# B&R Automation Studio project NewPendant_NG4_11_05_25A (part 5)

```c
	i = parCOOL_Tmo;
	strcpy(var[i].name , "Cool On/Off TimeOut");
	strcpy(var[i].enumTXT, "parCOOL_Tmo");
	var[i].PlcUnitIndx = unitIU;
	var[i].unitType = unitTime;
	var[i].DefaultUnit = UNIT_sec;
	var[i].precision = 1;
	cfg->Param[i].min = 0.0;
	cfg->Param[i].max = 5.0;
	cfg->Param[i].incrMin = 0.1;
	cfg->Param[i].incrMax = 1.0;
	cfg->Param[i].defaultVal = 3.0;
	var[i].segm = 0;

	///// INDX /////

	i = parINDX_StepDist;
	strcpy(var[i].name , "INDX Step Distance");
	strcpy(var[i].enumTXT, "parINDX_StepDist");
	var[i].PlcUnitIndx = unitIU;
	var[i].unitType = unitLength;
	var[i].DefaultUnit = UNIT_inch;
	var[i].precision = 1;
	cfg->Param[i].min = 0.0 * in_2_mm;
	cfg->Param[i].max = 200.0 * in_2_mm;
	cfg->Param[i].incrMin = 0.01 * in_2_mm;
	cfg->Param[i].incrMax = 1.0 * in_2_mm;
	cfg->Param[i].defaultVal = 4.5 * in_2_mm;
	var[i].segm = 0;

	i = parINDX_StepVel;
	strcpy(var[i].name , "INDX Step Vel");
	strcpy(var[i].enumTXT, "parINDX_StepVel");
	var[i].PlcUnitIndx = unitIU;
	var[i].unitType = unitPerc;
	var[i].DefaultUnit = UNIT_PERCENT;
	var[i].precision = 0;
	cfg->Param[i].min = 0.0;
	cfg->Param[i].max = 1.0;
	cfg->Param[i].incrMin = 0.01;
	cfg->Param[i].incrMax = 0.1;
	cfg->Param[i].defaultVal = 1.0;
	var[i].segm = 0;

	/*
	var[i].PlcUnitIndx = unitIU;
	var[i].unitType = unitSpeed;
	var[i].DefaultUnit = UNIT_inch_per_min;
	var[i].precision = 0;
	cfg->Param[i].min = 1.0 *  in_min_2_mm_s;
	cfg->Param[i].max = 10.0 *  in_min_2_mm_s;
	cfg->Param[i].incrMin = 0.1 * in_min_2_mm_s;
	cfg->Param[i].incrMax = 10.0 * cfg->Param[i].incrMin;
	cfg->Param[i].defaultVal = 3.0 * in_min_2_mm_s;
	var[i].segm = 0;
	*/

	i = parINDX_JogSpeedDirCntrl;
	strcpy(var[i].name , "INDX Jog Speed");
	strcpy(var[i].enumTXT, "parINDX_JogSpeedDirCntrl");
	var[i].PlcUnitIndx = unitIU;
	var[i].unitType = unitPerc;
	var[i].DefaultUnit = UNIT_PERCENT;
	var[i].precision = 0;
	cfg->Param[i].min = 0.0;
	cfg->Param[i].max = 1.0;
	cfg->Param[i].incrMin = 0.01;
	cfg->Param[i].incrMax = 0.1;
	cfg->Param[i].defaultVal = 1.0;
	var[i].segm = 0;

	i = parINDX_StepAfterBeats;
	strcpy(var[i].name , "Step After Beats");
	strcpy(var[i].enumTXT, "parINDX_StepAfterBeats");
	var[i].PlcUnitIndx = unitIU;
	var[i].unitType = unitIU;
	var[i].DefaultUnit = unitIU;
	var[i].precision = 0;
	cfg->Param[i].min = 0.0;
	cfg->Param[i].max = 99.0;
	cfg->Param[i].incrMin = 1.0;
	cfg->Param[i].incrMax = 1.0;
	cfg->Param[i].defaultVal = 0.0;
	var[i].segm = 0;

	//////  WRIST
	i = parWRST_JogSpeedDirCntrl;
	strcpy(var[i].name , "Weld Angle Jog Speed");
	strcpy(var[i].enumTXT, "parWRST_JogSpeedDirCntrl");
	var[i].PlcUnitIndx = unitIU;
	var[i].unitType = unitPerc;
	var[i].DefaultUnit = UNIT_PERCENT;
	var[i].precision = 1;
	cfg->Param[i].min = 0.0;
	cfg->Param[i].max = 1.0;
	cfg->Param[i].incrMin = 0.05;
	cfg->Param[i].incrMax = 0.1;
	cfg->Param[i].defaultVal = 0.75;
	var[i].segm = 0;

	//////  parTVL_POS_OFFSET
	i = parTVL_POS_OFFSET;
	strcpy(var[i].name , "TVL Pos Offset");
	strcpy(var[i].enumTXT, "parTVL_POS_OFFSET");
	var[i].PlcUnitIndx = unitIU;
	var[i].unitType = unitLength;
	var[i].DefaultUnit = UNIT_inch;
	var[i].precision = 1;
	cfg->Param[i].min = -200.0 * in_2_mm;
	cfg->Param[i].max = 200.0 * in_2_mm;
	cfg->Param[i].incrMin = 0.01 * in_2_mm;
	cfg->Param[i].incrMax = 1.0 * in_2_mm;
	cfg->Param[i].defaultVal = 0;
	var[i].segm = 0;

	i = parTVL_POS_PREDICT;
	strcpy(var[i].name , "TVL POS Predict Time");
	strcpy(var[i].enumTXT, "parTVL_POS_PREDICT");
	var[i].PlcUnitIndx = unitIU;
	var[i].unitType = unitTime;
	var[i].DefaultUnit = UNIT_sec;
	var[i].precision = 1;
	cfg->Param[i].min = 0.0;
	cfg->Param[i].max = 3.0;
	cfg->Param[i].incrMin = 0.1;
	cfg->Param[i].incrMax = 1.0;
	cfg->Param[i].defaultVal = 0.1;

	////////////////////////////////////

	i = parGEN_CalibDist;
	strcpy(var[i].name , "Calib Dist");
	strcpy(var[i].enumTXT, "parGEN_CalibDist");
	var[i].PlcUnitIndx = unitIU;
	var[i].unitType = unitLength;
	var[i].DefaultUnit = UNIT_inch;
	var[i].precision = 1;
	cfg->Param[i].min = 0.0;
	cfg->Param[i].max = 1000000;
	cfg->Param[i].incrMin = 0.254 *1;
	cfg->Param[i].incrMax = 25.4;
	cfg->Param[i].defaultVal = 0.0;
	var[i].segm = 0;

	i = parGEN_CalibDist_2;
	strcpy(var[i].name , "Calib Dist 2");
	strcpy(var[i].enumTXT, "parGEN_CalibDist_2");
	var[i].PlcUnitIndx = unitIU;
	var[i].unitType = unitLength;
	var[i].DefaultUnit = UNIT_inch;
	var[i].precision = 1;
	cfg->Param[i].min = 0.0;
	cfg->Param[i].max = 1000000;
	cfg->Param[i].incrMin = 0.254 *1;
	cfg->Param[i].incrMax = 25.4;
	cfg->Param[i].defaultVal = 0.0;
	var[i].segm = 0;

	i = parGEN_CalibDist1;
	strcpy(var[i].name , "Calib Dist1");
	strcpy(var[i].enumTXT, "parGEN_CalibDist1");
	var[i].PlcUnitIndx = unitIU;
	var[i].unitType = unitLength;
	var[i].DefaultUnit = UNIT_inch;
	var[i].precision = 1;
	cfg->Param[i].min = 0.0;
	cfg->Param[i].max = 1000000;
	cfg->Param[i].incrMin = 0.254 *1;
	cfg->Param[i].incrMax = 25.4;
	cfg->Param[i].defaultVal = 0.0;
	var[i].segm = 0;

	i = parGEN_CalibDist2;
	strcpy(var[i].name , "Calib Dist2");
	strcpy(var[i].enumTXT, "parGEN_CalibDist2");
	var[i].PlcUnitIndx = unitIU;
	var[i].unitType = unitLength;
	var[i].DefaultUnit = UNIT_inch;
	var[i].precision = 1;
	cfg->Param[i].min = 0.0;
	cfg->Param[i].max = 1000000;
	cfg->Param[i].incrMin = 0.254 *1;
	cfg->Param[i].incrMax = 25.4;
	cfg->Param[i].defaultVal = 0.0;
	var[i].segm = 0;

	i = parGEN_CalibDist3;
	strcpy(var[i].name , "Calib Dist3");
	strcpy(var[i].enumTXT, "parGEN_CalibDist3");
	var[i].PlcUnitIndx = unitIU;
	var[i].unitType = unitLength;
	var[i].DefaultUnit = UNIT_inch;
	var[i].precision = 1;
	cfg->Param[i].min = 0.0;
	cfg->Param[i].max = 1000000;
	cfg->Param[i].incrMin = 0.254 *1;
	cfg->Param[i].incrMax = 25.4;
	cfg->Param[i].defaultVal = 0.0;
	var[i].segm = 0;

	i = parGEN_CalibDist4;
	strcpy(var[i].name , "Calib Dist4");
	strcpy(var[i].enumTXT, "parGEN_CalibDist4");
	var[i].PlcUnitIndx = unitIU;
	var[i].unitType = unitLength;
	var[i].DefaultUnit = UNIT_inch;
	var[i].precision = 1;
	cfg->Param[i].min = 0.0;
	cfg->Param[i].max = 1000000;
	cfg->Param[i].incrMin = 0.254 *1;
	cfg->Param[i].incrMax = 25.4;
	cfg->Param[i].defaultVal = 0.0;
	var[i].segm = 0;

	i = parGEN_CalibTime;
	strcpy(var[i].name , "Calib Time");
	strcpy(var[i].enumTXT, "parGEN_CalibTime");
	var[i].PlcUnitIndx = unitIU;
	var[i].unitType = unitTime;
	var[i].DefaultUnit = UNIT_sec;
	var[i].precision = 1;
	cfg->Param[i].min = 0.0;
	cfg->Param[i].max = 1000000000.0;
	cfg->Param[i].incrMin = 0.05;
	cfg->Param[i].incrMax = 10.0;
	cfg->Param[i].defaultVal = 0.0;
	var[i].segm = 0;

	i = parGEN_CalibTime1;
	strcpy(var[i].name , "Calib Time1");
	strcpy(var[i].enumTXT, "parGEN_CalibTime1");
	var[i].PlcUnitIndx = unitIU;
	var[i].unitType = unitTime;
	var[i].DefaultUnit = UNIT_sec;
	var[i].precision = 1;
	cfg->Param[i].min = 0.0;
	cfg->Param[i].max = 1000000000.0;
	cfg->Param[i].incrMin = 0.05;
	cfg->Param[i].incrMax = 10.0;
	cfg->Param[i].defaultVal = 0.0;
	var[i].segm = 0;

	i = parGEN_CalibTime2;
	strcpy(var[i].name , "Calib Time2");
	strcpy(var[i].enumTXT, "parGEN_CalibTime2");
	var[i].PlcUnitIndx = unitIU;
	var[i].unitType = unitTime;
	var[i].DefaultUnit = UNIT_sec;
	var[i].precision = 1;
	cfg->Param[i].min = 0.0;
	cfg->Param[i].max = 1000000000.0;
	cfg->Param[i].incrMin = 0.05;
	cfg->Param[i].incrMax = 10.0;
	cfg->Param[i].defaultVal = 0.0;
	var[i].segm = 0;

	i = parGEN_CalibTime3;
	strcpy(var[i].name , "Calib Time3");
	strcpy(var[i].enumTXT, "parGEN_CalibTime3");
	var[i].PlcUnitIndx = unitIU;
	var[i].unitType = unitTime;
	var[i].DefaultUnit = UNIT_sec;
	var[i].precision = 1;
	cfg->Param[i].min = 0.0;
	cfg->Param[i].max = 1000000000.0;
	cfg->Param[i].incrMin = 0.05;
	cfg->Param[i].incrMax = 10.0;
	cfg->Param[i].defaultVal = 0.0;
	var[i].segm = 0;

	i = parGEN_CalibAmp1;
	strcpy(var[i].name , "GEN Calib Amp 1");
	strcpy(var[i].enumTXT, "parGEN_CalibAmp1");
	var[i].PlcUnitIndx = unitIU;
	var[i].unitType = unitAmp;
	var[i].DefaultUnit = UNIT_Amp;
	var[i].precision = 0;
	cfg->Param[i].min = 1.0;
	cfg->Param[i].max = 500.0;
	cfg->Param[i].incrMin = 1.0;
	cfg->Param[i].incrMax = 10.0;
	cfg->Param[i].defaultVal = 25.0;
	var[i].segm = 0;

	i = parGEN_CalibAmp2;
	strcpy(var[i].name , "GEN Calib Amp 2");
	strcpy(var[i].enumTXT, "parGEN_CalibAmp2");
	var[i].PlcUnitIndx = unitIU;
	var[i].unitType = unitAmp;
	var[i].DefaultUnit = UNIT_Amp;
	var[i].precision = 0;
	cfg->Param[i].min = 1.0;
	cfg->Param[i].max = 500.0;
	cfg->Param[i].incrMin = 1.0;
	cfg->Param[i].incrMax = 10.0;
	cfg->Param[i].defaultVal = 25.0;
	var[i].segm = 0;

	i = parGEN_CalibTime4;
	strcpy(var[i].name , "Calib Time4");
	strcpy(var[i].enumTXT, "parGEN_CalibTime4");
	var[i].PlcUnitIndx = unitIU;
	var[i].unitType = unitTime;
	var[i].DefaultUnit = UNIT_sec;
	var[i].precision = 1;
	cfg->Param[i].min = 0.0;
	cfg->Param[i].max = 1000000000.0;
	cfg->Param[i].incrMin = 0.05;
	cfg->Param[i].incrMax = 10.0;
	cfg->Param[i].defaultVal = 0.0;
	var[i].segm = 0;

	i = parGEN_AmpRead;
	strcpy(var[i].name , "Amp Meas.");
	strcpy(var[i].enumTXT, "parGEN_AmpRead");
	var[i].PlcUnitIndx = unitIU;
	var[i].unitType = unitAmp;
	var[i].DefaultUnit = UNIT_Amp;
	var[i].precision = 0;
	cfg->Param[i].min = 5.0;
	cfg->Param[i].max = 200.0;
	cfg->Param[i].incrMin = 1.0;
	cfg->Param[i].incrMax = 10.0;
	cfg->Param[i].defaultVal = 50.0;
	var[i].segm = 0;

	i = parGEN_WeldProgramRepeat;
	strcpy(var[i].name , "Weld Program Repeat");
	strcpy(var[i].enumTXT, "parGEN_WeldProgramRepeat");
	var[i].PlcUnitIndx = unitIU;
	var[i].unitType = unitIU;
	var[i].DefaultUnit = unitIU;
	var[i].precision = 0;
	cfg->Param[i].min = 0.0;
	cfg->Param[i].max = 99.0;
	cfg->Param[i].incrMin = 1.0;
	cfg->Param[i].incrMax = 1.0;
	cfg->Param[i].defaultVal = 0.0;
	var[i].segm = 0;

	i = parGEN_RadSpeed_Boost;
	strcpy(var[i].name , "TVL Radius Vel Boost");
	strcpy(var[i].enumTXT, "parGEN_RadSpeed_Boost");
	var[i].PlcUnitIndx = unitIU;
	var[i].unitType = unitPerc;
	var[i].DefaultUnit = UNIT_PERCENT;
	var[i].precision = 1;
	cfg->Param[i].min = 0.0;
	cfg->Param[i].max = 10.0;
	cfg->Param[i].incrMin = 0.05;
	cfg->Param[i].incrMax = 0.1;
	cfg->Param[i].defaultVal = 2.0;
	var[i].segm = 0;

	i = parGEN_Radius;
	strcpy(var[i].name , "Pole Radius");
	strcpy(var[i].enumTXT, "parGEN_Radius");
	var[i].PlcUnitIndx = unitIU;
	var[i].unitType = unitLength;
	var[i].DefaultUnit = UNIT_inch;
	var[i].precision = 1;
	cfg->Param[i].min = 0.0;
	cfg->Param[i].max = 1000000;
	cfg->Param[i].incrMin = 0.254 *1;
	cfg->Param[i].incrMax = 25.4;
	cfg->Param[i].defaultVal = 0.0;
	var[i].segm = 0;

	/////////////////////////////////////
	////////   Scaled variables

	i = varCurTVL_Vel;
	strcpy(var[i].enumTXT, "varCurTVL_Vel");
	strcpy(var[i].name , "TVL Vel 1FBK");
	var[i].pfVal = &Process[PROC_TVL].Fbk[0];
	strcpy(var[i].VarName , "Process[0].Fbk[0]");
	var[i].type = VAR_READONLY;
	var[i].PlcUnitIndx = unitIU;
	var[i].unitType = unitSpeed;
	var[i].DefaultUnit = UNIT_inch_per_min;
	var[i].precision = 0;

	i = varCurTVL_Vel_Calc;
	strcpy(var[i].enumTXT, "varCurTVL_Vel_Calc");
	strcpy(var[i].name , "TVL Vel FBK Calc");
	var[i].pfVal = &Process[PROC_TVL].Fbk[4];
	strcpy(var[i].VarName , "Process[0].Fbk[4]");
	var[i].type = VAR_READONLY;
	var[i].PlcUnitIndx = unitIU;
	var[i].unitType = unitSpeed;
	var[i].DefaultUnit = UNIT_inch_per_min;
	var[i].precision = 2;

	i = varTVL_Vel_Cmd;
	strcpy(var[i].enumTXT, "varTVL_Vel_Cmd");
	strcpy(var[i].name , "TVL Vel Cmd");
	var[i].pfVal = &Process[PROC_TVL].Fbk[1];
	strcpy(var[i].VarName , "Process[0].Fbk[1]");
	var[i].type = VAR_READONLY;
	var[i].PlcUnitIndx = unitIU;
	var[i].unitType = unitSpeed;
	var[i].DefaultUnit = UNIT_inch_per_min;
	var[i].precision = 0;

	i = varCurWF_Vel;
	strcpy(var[i].enumTXT, "varCurWF_Vel");
	strcpy(var[i].name , "WF Vel FBK");
	var[i].pfVal = &Process[PROC_WIRE_FEED].Fbk[0];
	strcpy(var[i].VarName , "Process[3].Fbk[0]");
	var[i].type = VAR_READONLY;
	var[i].PlcUnitIndx = unitIU;
	var[i].unitType = unitSpeed;
	var[i].DefaultUnit = UNIT_inch_per_min;
	var[i].precision = 0;

	i = varWF_Vel_Cmd;
	strcpy(var[i].enumTXT, "varWF_Vel_Cmd");
	strcpy(var[i].name , "WF Vel Cmd");
	var[i].pfVal = &Process[PROC_WIRE_FEED].Fbk[1];
	strcpy(var[i].VarName , "Process[3].Fbk[1]");
	var[i].type = VAR_READONLY;
	var[i].PlcUnitIndx = unitIU;
	var[i].unitType = unitSpeed;
	var[i].DefaultUnit = UNIT_inch_per_min;
	var[i].precision = 0;

	i = varCurWFDist;
	strcpy(var[i].enumTXT, "varCurWFDist");
	strcpy(var[i].name , "act WF Len");
	var[i].pfVal = &Process[PROC_WIRE_FEED].Fbk[4];
	strcpy(var[i].VarName , "Process[3].Fbk[4]");
	var[i].type = VAR_READONLY;
	var[i].PlcUnitIndx = unitIU;
	var[i].unitType = unitLength;
	var[i].DefaultUnit = UNIT_inch;
	var[i].precision = 0;

	i = varCurWP_Vel;
	strcpy(var[i].enumTXT, "varCurWP_Vel");
	strcpy(var[i].name , "WP Freq FBK");
	var[i].pfVal = &Process[PROC_WIRE_PULSE].Fbk[0];
	strcpy(var[i].VarName , "Process[4].Fbk[0]");
	var[i].type = VAR_READONLY;
	var[i].PlcUnitIndx = unitIU;
	var[i].unitType = unitFreq;
	var[i].DefaultUnit = UNIT_Hz;
	var[i].precision = 1;

	i = varWP_Vel_Cmd;
	strcpy(var[i].enumTXT, "varWP_Vel_Cmd");
	strcpy(var[i].name , "WP Freq Cmd");
	var[i].pfVal = &Process[PROC_WIRE_PULSE].Fbk[1];
	strcpy(var[i].VarName , "Process[4].Fbk[1]");
	var[i].type = VAR_READONLY;
	var[i].PlcUnitIndx = unitIU;
	var[i].unitType = unitFreq;
	var[i].DefaultUnit = UNIT_Hz;
	var[i].precision = 1;

	i = varCurArc_Volt;
	strcpy(var[i].enumTXT, "varCurArc_Volt");
	strcpy(var[i].name , "Arc Volt FBK");
	var[i].pfVal = &Process[PROC_AVC].Fbk[0];
	strcpy(var[i].VarName , "Process[2].Fbk[0]");
	var[i].type = VAR_READONLY;
	var[i].PlcUnitIndx = unitIU;
	var[i].unitType = unitVolt;
	var[i].DefaultUnit = UNIT_Volt;
	var[i].precision = 1;

	i = varArc_Volt_Cmd;
	strcpy(var[i].enumTXT, "varArc_Volt_Cmd");
	strcpy(var[i].name , "Arc Volt Cmd");
	var[i].pfVal = &Process[PROC_AVC].Fbk[1];
	strcpy(var[i].VarName , "Process[2].Fbk[1]");
	var[i].type = VAR_READONLY;
	var[i].PlcUnitIndx = unitIU;
	var[i].unitType = unitVolt;
	var[i].DefaultUnit = UNIT_Volt;
	var[i].precision = 1;

	i = varCurTIG_Amp;
	strcpy(var[i].enumTXT, "varCurTIG_Amp");
	strcpy(var[i].name , "TIG Amp FBK");
	var[i].pfVal = &Process[PROC_TIG_PS].Fbk[0];
	strcpy(var[i].VarName , "Process[5].Fbk[0]");
	var[i].type = VAR_READONLY;
	var[i].PlcUnitIndx = unitIU;
	var[i].unitType = unitAmp;
	var[i].DefaultUnit = UNIT_Amp;
	var[i].precision = 1;

	i = varTIG_Amp_Cmd;
	strcpy(var[i].enumTXT, "varTIG_Amp_Cmd");
	strcpy(var[i].name , "TIG Amp CMD");
	var[i].pfVal = &Process[PROC_TIG_PS].Fbk[1];
	strcpy(var[i].VarName , "Process[5].Fbk[1]");
	var[i].type = VAR_READONLY;
	var[i].PlcUnitIndx = unitIU;
	var[i].unitType = unitAmp;
	var[i].DefaultUnit = UNIT_Amp;
	var[i].precision = 0;

	i = varCurHW_Amp;
	strcpy(var[i].enumTXT, "varCurHW_Amp");
	strcpy(var[i].name , "HW Amp FBK");
	var[i].pfVal = &Process[PROC_HW_PS].Fbk[0];
	strcpy(var[i].VarName , "Process[6].Fbk[0]");
	var[i].type = VAR_READONLY;
	var[i].PlcUnitIndx = unitIU;
	var[i].unitType = unitAmp;
	var[i].DefaultUnit = UNIT_Amp;
	var[i].precision = 0;

	i = varHW_Amp_Cmd;
	strcpy(var[i].enumTXT, "varHW_Amp_Cmd");
	strcpy(var[i].name , "HW Amp CMD");
	var[i].pfVal = &Process[PROC_HW_PS].Fbk[1];
	strcpy(var[i].VarName , "Process[6].Fbk[1]");
	var[i].type = VAR_READONLY;
	var[i].PlcUnitIndx = unitIU;
	var[i].unitType = unitAmp;
	var[i].DefaultUnit = UNIT_Amp;
	var[i].precision = 0;

	i = varCurHW_Volt; // new
	strcpy(var[i].enumTXT, "varCurHW_Volt");
	strcpy(var[i].name , "HW Volt FBK");
	var[i].pfVal = &Process[PROC_HW_PS].Fbk[2];
	strcpy(var[i].VarName , "Process[6].Fbk[2]");
	var[i].type = VAR_READONLY;
	var[i].PlcUnitIndx = unitIU;
	var[i].unitType = unitVolt;
	var[i].DefaultUnit = UNIT_Volt;
	var[i].precision = 1;

	i = varHW_Volt_Cmd; // new
	strcpy(var[i].enumTXT, "varHW_Volt_Cmd");
	strcpy(var[i].name , "HW Volt CMD");
	var[i].pfVal = &Process[PROC_HW_PS].Fbk[3];
	strcpy(var[i].VarName , "Process[6].Fbk[3]");
	var[i].type = VAR_READONLY;
	var[i].PlcUnitIndx = unitIU;
	var[i].unitType = unitVolt;
	var[i].DefaultUnit = UNIT_Volt;
	var[i].precision = 1;

	i = varOSC_CurPos;
	strcpy(var[i].enumTXT, "varOSC_CurPos");
	strcpy(var[i].name , "act OSC Pos");
	var[i].pfVal = &Process[PROC_OSC].Fbk[0];
	strcpy(var[i].VarName , "Process[1].Fbk[0]");
	var[i].type = VAR_READONLY;
	var[i].PlcUnitIndx = unitIU;
	var[i].unitType = unitLength;
	var[i].DefaultUnit = UNIT_inch;
	var[i].precision = 1;

	i = varOSC_Centr;
	strcpy(var[i].enumTXT, "varOSC_Centr");
	strcpy(var[i].name , "act OSC Centr");
	var[i].pfVal = &Process[PROC_OSC].Fbk[1];
	strcpy(var[i].VarName , "Process[1].Fbk[1]");
	var[i].type = VAR_READONLY;
	var[i].PlcUnitIndx = unitIU;
	var[i].unitType = unitLength;
	var[i].DefaultUnit = UNIT_inch;
	var[i].precision = 1;

	i = varOSC_CurRawPos;
	strcpy(var[i].enumTXT, "varOSC_CurRawPos");
	strcpy(var[i].name , "act OSC Pos");
	var[i].pfVal = &Process[PROC_OSC].Fbk[2];
	strcpy(var[i].VarName , "Process[1].Fbk[2]");
	var[i].type = VAR_READONLY;
	var[i].PlcUnitIndx = unitIU;
	var[i].unitType = unitLength;
	var[i].DefaultUnit = UNIT_inch;
	var[i].precision = 2;

	i = varOSC_Amplit_Cmd;
	strcpy(var[i].enumTXT, "varOSC_Amplit_Cmd");
	strcpy(var[i].name , "OSC Amplit Cmd");
	var[i].pfVal = &Process[PROC_OSC].Fbk[3];
	strcpy(var[i].VarName , "Process[1].Fbk[3]");
	var[i].type = VAR_READONLY;
	var[i].PlcUnitIndx = unitIU;
	var[i].unitType = unitLength;
	var[i].DefaultUnit = UNIT_inch;
	var[i].precision = 1;

	i = varOSC_curExcurTm;
	strcpy(var[i].enumTXT, "varOSC_curExcurTm");
	strcpy(var[i].name , "act Excur Tm");
	var[i].pfVal = &Process[PROC_OSC].Fbk[4];
	strcpy(var[i].VarName , "Process[1].Fbk[4]");
	var[i].type = VAR_READONLY;
	var[i].PlcUnitIndx = unitIU;
	var[i].unitType = unitTime;
	var[i].DefaultUnit = UNIT_sec;
	var[i].precision = 1;

	i = varOSC_ExcurTm_Cmd;
	strcpy(var[i].enumTXT, "varOSC_ExcurTm_Cmd");
	strcpy(var[i].name , "OSC Excur Tm Cmd");
	var[i].pfVal = &Process[PROC_OSC].Fbk[5];
	strcpy(var[i].VarName , "Process[1].Fbk[5]");
	var[i].type = VAR_READONLY;
	var[i].PlcUnitIndx = unitIU;
	var[i].unitType = unitTime;
	var[i].DefaultUnit = UNIT_sec;
	var[i].precision = 1;

	i = varOSC_Dwell_In_Cmd;
	strcpy(var[i].enumTXT, "varOSC_Dwell_In_Cmd");
	strcpy(var[i].name , "varOSC Dwell In Cmd");
	var[i].pfVal = &Process[PROC_OSC].Fbk[6];
	strcpy(var[i].VarName , "Process[1].Fbk[6]");
	var[i].type = VAR_READONLY;
	var[i].PlcUnitIndx = unitIU;
	var[i].unitType = unitTime;
	var[i].DefaultUnit = UNIT_sec;
	var[i].precision = 1;

	i = varOSC_Dwell_Out_Cmd;
	strcpy(var[i].enumTXT, "varOSC_Dwell_Out_Cmd");
	strcpy(var[i].name , "Dwell_Out_Cmd Cmd");
	var[i].pfVal = &Process[PROC_OSC].Fbk[7];
	strcpy(var[i].VarName , "Process[1].Fbk[7]");
	var[i].type = VAR_READONLY;
	var[i].PlcUnitIndx = unitIU;
	var[i].unitType = unitTime;
	var[i].DefaultUnit = UNIT_sec;
	var[i].precision = 1;

	i = varINDX_A_Pos;
	strcpy(var[i].enumTXT, "varINDX_A_Pos");
	strcpy(var[i].name , "act Indx A Pos");
	var[i].pfVal = &Process[PROC_INDX].Fbk[0];
	strcpy(var[i].VarName , "Process[10].Fbk[0]");
	var[i].type = VAR_READONLY;
	var[i].PlcUnitIndx = unitIU;
	var[i].unitType = unitLength;
	var[i].DefaultUnit = UNIT_inch;
	var[i].precision = 2;

	i = varINDX_B_Pos;
	strcpy(var[i].enumTXT, "varINDX_B_Pos");
	strcpy(var[i].name , "act Indx B Pos");
	var[i].pfVal = &Process[PROC_INDX].Fbk[1];
	strcpy(var[i].VarName , "Process[10].Fbk[1]");
	var[i].type = VAR_READONLY;
	var[i].PlcUnitIndx = unitIU;
	var[i].unitType = unitLength;
	var[i].DefaultUnit = UNIT_inch;
	var[i].precision = 2;

	i = varINDX_Dif_Pos;
	strcpy(var[i].enumTXT, "varINDX_Dif_Pos");
	strcpy(var[i].name , "act Indx Dif Pos");
	var[i].pfVal = &Process[PROC_INDX].Fbk[2];
	strcpy(var[i].VarName , "Process[10].Fbk[2]");
	var[i].type = VAR_READONLY;
	var[i].PlcUnitIndx = unitIU;
	var[i].unitType = unitLength;
	var[i].DefaultUnit = UNIT_inch;
	var[i].precision = 3;

	i = varGlobTimer;
	strcpy(var[i].enumTXT, "varGlobTimer");
	strcpy(var[i].name , "Timer");
	var[i].pfVal = &GlobalTimer;
	strcpy(var[i].VarName , "GlobalTimer");
	var[i].type = VAR_READONLY;
	var[i].PlcUnitIndx = unitIU;
	var[i].unitType = unitTime;
	var[i].DefaultUnit = UNIT_sec;
	var[i].precision = 0;

	////////////////////////////

	i = parENUM_OSC_CAM;
	strcpy(cfg->EnumVar[i].enumTXT , "parENUM_OSC_CAM");
	strcpy(cfg->EnumVar[i].name , "OSC Cam Type ");
	cfg->EnumVar[i].TxtIndx = resTXT_OSC_CAM;
	cfg->EnumVar[i].segm = 0;
	cfg->Param_ENUM[i].defaultVal = 1;
	cfg->Param_ENUM[i].min = 0;
	cfg->Param_ENUM[i].max = CAM_NUM-1;

	i = parENUM_WeldProgramLinkMode;
	strcpy(cfg->EnumVar[i].enumTXT , "parENUM_WeldProgramLinkMode");
	strcpy(cfg->EnumVar[i].name , "Load Next Program ");
	cfg->EnumVar[i].TxtIndx = resWelProgramLinkMode;
	cfg->EnumVar[i].segm = 0;
	cfg->Param_ENUM[i].defaultVal = 0;
	cfg->Param_ENUM[i].min = 0;
	cfg->Param_ENUM[i].max = 1;

	i= parENUM_PathMode;
	strcpy(cfg->EnumVar[i].enumTXT , "parENUM_PathMode");
	strcpy(cfg->EnumVar[i].name , "Change Head at the end ");
	cfg->EnumVar[i].TxtIndx = resPathMode;
	cfg->EnumVar[i].segm = 0;
	cfg->Param_ENUM[i].defaultVal = 0;
	cfg->Param_ENUM[i].min = 0;
	cfg->Param_ENUM[i].max = 1;

	i= parENUM_TVL_MODE;
	strcpy(cfg->EnumVar[i].enumTXT , "parENUM_TVL_MODE");
	strcpy(cfg->EnumVar[i].name , "TVL Enc Mode");
	cfg->EnumVar[i].TxtIndx = resTVLMode;
	cfg->EnumVar[i].segm = 0;
	cfg->Param_ENUM[i].defaultVal = 0;
	cfg->Param_ENUM[i].min = 0;
	cfg->Param_ENUM[i].max = 3;

	i= parENUM_TVL_SYN_MODE;
	strcpy(cfg->EnumVar[i].enumTXT , "parENUM_TVL_SYN_MODE");
	strcpy(cfg->EnumVar[i].name , "TVL Synch Mode");
	cfg->EnumVar[i].TxtIndx = resSYNCOption; // Chris add this parameter to enum
	cfg->EnumVar[i].segm = 0;
	cfg->Param_ENUM[i].defaultVal = 0;
	cfg->Param_ENUM[i].min = 0;
	cfg->Param_ENUM[i].max = 2;

	i= parENUM_WF_SYN_MODE;
	strcpy(cfg->EnumVar[i].enumTXT , "parENUM_WF_SYN_MODE");
	strcpy(cfg->EnumVar[i].name , "WF Synch Mode");
	cfg->EnumVar[i].TxtIndx = resSYNCOption;
	cfg->EnumVar[i].segm = 0;
	cfg->Param_ENUM[i].defaultVal = 0;
	cfg->Param_ENUM[i].min = 0;
	cfg->Param_ENUM[i].max = 2;

	i= parENUM_WP_SYN_MODE;
	strcpy(cfg->EnumVar[i].enumTXT , "parENUM_WP_SYN_MODE");
	strcpy(cfg->EnumVar[i].name , "WP Synch Mode");
	cfg->EnumVar[i].TxtIndx = resSYNCOption;
	cfg->EnumVar[i].segm = 0;
	cfg->Param_ENUM[i].defaultVal = 0;
	cfg->Param_ENUM[i].min = 0;
	cfg->Param_ENUM[i].max = 2;

	/*
	i = parENUM_WeldProgramCase;
	strcpy(cfg->EnumVar[i].enumTXT , ""); // Use as a spare
	//strcpy(cfg->EnumVar[i].enumTXT , "parENUM_WeldProgramCase");
	cfg->EnumVar[i].TxtIndx = resWeldProgramCase;
	cfg->EnumVar[i].segm = 0;
	cfg->Param_ENUM[i].defaultVal = 0;
	cfg->Param_ENUM[i].min = 0;
	cfg->Param_ENUM[i].max = 5;
	*/

	i = parENUM_AVC_Mode;
	strcpy(cfg->EnumVar[i].enumTXT , "parENUM_AVC_Mode");
	strcpy(cfg->EnumVar[i].name , "AVC Type ");
	cfg->EnumVar[i].TxtIndx = resAVCMode;
	cfg->EnumVar[i].segm = 0;
	cfg->Param_ENUM[i].defaultVal = 0;
	cfg->Param_ENUM[i].min = 0;
	cfg->Param_ENUM[i].max = 3;

	i = parENUM_TIG_Mode;
	strcpy(cfg->EnumVar[i].enumTXT , "parENUM_TIG_Mode");
	strcpy(cfg->EnumVar[i].name , "TIG PS Mode ");
	cfg->EnumVar[i].TxtIndx = resTIGMode;
	cfg->EnumVar[i].segm = 0;
	cfg->Param_ENUM[i].defaultVal = 0;
	cfg->Param_ENUM[i].min = 0;
	cfg->Param_ENUM[i].max = 3;

	i = parENUM_TIG_Cal_Mode;
	strcpy(cfg->EnumVar[i].enumTXT , "parENUM_TIG_Cal_Mode");
	strcpy(cfg->EnumVar[i].name , "TIG PS Cal. Mode ");
	cfg->EnumVar[i].TxtIndx = resTigCalMode;
	cfg->EnumVar[i].segm = 0;
	cfg->Param_ENUM[i].defaultVal = 0;
	cfg->Param_ENUM[i].min = 0;
	cfg->Param_ENUM[i].max = 1;

	i = parENUM_WF_WP_Relation;
	strcpy(cfg->EnumVar[i].enumTXT , "parENUM_WF_WP_Relation");
	strcpy(cfg->EnumVar[i].name , "Relation between WF and WP");
	cfg->EnumVar[i].TxtIndx = resTXT_ON_OFF;
	cfg->EnumVar[i].segm = 0;
	cfg->Param_ENUM[i].defaultVal = 0;
	cfg->Param_ENUM[i].min = 0;
	cfg->Param_ENUM[i].max = 1;

	i = parENUM_ARCLINK_MODE;
	strcpy(cfg->EnumVar[i].enumTXT , "parENUM_ARCLINK_MODE");
	strcpy(cfg->EnumVar[i].name , "ARcLink ");
	cfg->EnumVar[i].TxtIndx = resTXT_ON_OFF;
	cfg->EnumVar[i].segm = 0;
	cfg->Param_ENUM[i].defaultVal = 0;
	cfg->Param_ENUM[i].min = 0;
	cfg->Param_ENUM[i].max = 1;

	i = parENUM_OSC_Mode;
	strcpy(cfg->EnumVar[i].enumTXT , "parENUM_OSC_Mode");
	strcpy(cfg->EnumVar[i].name , "OSC Mode ");
	cfg->EnumVar[i].TxtIndx = resTXT_OSC_Mode;
	cfg->EnumVar[i].segm = 0;
	cfg->Param_ENUM[i].defaultVal = 0;
	cfg->Param_ENUM[i].min = 0;
	cfg->Param_ENUM[i].max = 3;

	i = parENUM_OSC_Synch;
	strcpy(cfg->EnumVar[i].enumTXT , "parENUM_OSC_Synch");
	strcpy(cfg->EnumVar[i].name , "OSC Indx Synch ");
	cfg->EnumVar[i].TxtIndx = resTXT_OSC_Synch;
	cfg->EnumVar[i].segm = 0;
	cfg->Param_ENUM[i].defaultVal = 0;
	cfg->Param_ENUM[i].min = 0;
	cfg->Param_ENUM[i].max = 4;

	i = parENUM_WF_AUX;
	strcpy(cfg->EnumVar[i].enumTXT , "parENUM_WF_AUX");
	strcpy(cfg->EnumVar[i].name , "parENUM_WF_AUX");
	cfg->EnumVar[i].TxtIndx = resTXT_WF_AUX;
	cfg->EnumVar[i].segm = 0;
	cfg->Param_ENUM[i].defaultVal = 0;
	cfg->Param_ENUM[i].min = 0;
	cfg->Param_ENUM[i].max = 2;

	///////Int Variable    //////////

	i = parINT_NumZone;
	strcpy(cfg->IntVar[i].enumTXT , "parINT_NumZone");
	strcpy(cfg->IntVar[i].name , 	"Segments per Travel");
	cfg->IntVar[i].pVal = &curCfg->Param_INT[parINT_NumZone].val[0];
	strcpy(cfg->IntVar[i].VarName , "CurCfg.Param_INT[0].val[0]"); //this is for Android
	cfg->IntVar[i].DefaultVal = 1;
	cfg->IntVar[i].Min = 1;
	cfg->IntVar[i].Max = 1000;
	cfg->IntVar[i].segm = 0;

	i = varINT_PIN_PER_ROT;
	strcpy(cfg->IntVar[i].enumTXT , "varINT_PIN_PER_ROT");
	strcpy(cfg->IntVar[i].name , 	"Pins per 360 degree");
	cfg->IntVar[i].pVal = &calib->GenSetup[SETUP_PIN_PER_ROT];
	strcpy(cfg->IntVar[i].VarName , "CurCalib.GenSetup[0]"); //this is for Android
	cfg->IntVar[i].Min = 1;
	cfg->IntVar[i].Max = 1000;

	i = varINT_SEGM_NO;
	strcpy(cfg->IntVar[i].enumTXT , "varINT_SEGM_NO");
	strcpy(cfg->IntVar[i].name , 	"Segments Number");
	cfg->IntVar[i].pVal = &calib->GenSetup[SETUP_SEGM_NO];
	strcpy(cfg->IntVar[i].VarName , "CurCalib.GenSetup[1]"); //this is for Android
	cfg->IntVar[i].Min = 1;
	cfg->IntVar[i].Max = 1000;

	/*
	i = varINT_ZONE_NO;
	strcpy(cfg->IntVar[i].enumTXT , "varINT_ZONE_NO");
	cfg->IntVar[i].pVal = &calib->GenSetup[SETUP_ZONE_NO];
	strcpy(cfg->IntVar[i].VarName , "CurCalib.GenSetup[2]"); //this is for Android
	cfg->IntVar[i].Min = 1;
	cfg->IntVar[i].Max = 1000;

	i= varINT_curSegm;
	strcpy(cfg->IntVar[i].enumTXT , "varINT_curSegm");
	strcpy(cfg->IntVar[i].name , 	"Current Pin");
	cfg->IntVar[i].pVal = &m->curSegm[HEAD_SEGM];
	strcpy(cfg->IntVar[i].VarName , "Master[0].curSegm[3]"); //this is for Android
	cfg->IntVar[i].Min = 1;
	cfg->IntVar[i].Max = 1000;
	*/

	i = varINT_curZone;
	strcpy(cfg->IntVar[i].enumTXT , "varINT_curZone");
	strcpy(cfg->IntVar[i].name , 	"Current Segment");
	cfg->IntVar[i].pVal = &m->curSegm[ZONE];
	strcpy(cfg->IntVar[i].VarName , "Master[0].curSegm[1]"); //this is for Android
	cfg->IntVar[i].Min = 1;
	cfg->IntVar[i].Max = 1000;

	i = varINT_StartPos;
	strcpy(cfg->IntVar[i].enumTXT , "varINT_StartPos");
	strcpy(cfg->IntVar[i].name , 	"Start Position");
	cfg->IntVar[i].pVal = &StartPos;
	strcpy(cfg->IntVar[i].VarName , "StartPos"); //this is for Android
	cfg->IntVar[i].Min = -32767;
	cfg->IntVar[i].Max = 32767;

	i = varINT_FinalPos;
	strcpy(cfg->IntVar[i].enumTXT , "varINT_FinalPos");
	strcpy(cfg->IntVar[i].name , 	"Target Position");
	cfg->IntVar[i].pVal = &FinalPos;
	strcpy(cfg->IntVar[i].VarName , "FinalPos"); //this is for Android
	cfg->IntVar[i].Min = -32767;
	cfg->IntVar[i].Max = 32767;

	i = varINT_CurTVLPos;
	strcpy(cfg->IntVar[i].enumTXT , "varINT_CurTVLPos");
	strcpy(cfg->IntVar[i].name , 	"Current TVL Position");
	cfg->IntVar[i].pVal = &m->curSegm[ACT_TVL_DIST];
	strcpy(cfg->IntVar[i].VarName , "Master[0].curSegm[4]"); //this is for Android
	cfg->IntVar[i].Min = -32767;
	cfg->IntVar[i].Max = 32767;

	/// Strings
	i = parSTRING_FreeTXT;
	strcpy(cfg->StringVar[i].enumTXT , "parSTRING_FreeTXT");
	strcpy(cfg->StringVar[i].name, "FreeText");
	cfg->Param_STR[i].len = 5;
	if(strlen(curCfg->Param_STR[i].str) == 0 )
		strcpy(curCfg->Param_STR[i].str , "12345");

	i = varSTRING_NextProgramName;
	strcpy(cfg->StringVar[i].enumTXT , "varSTRING_NextProgramName");
	strcpy(cfg->StringVar[i].name, "Next Program Name");
	cfg->StringVar[i].pStr = curCfg->NextProgramName;
	strcpy(cfg->StringVar[i].VarName , "CurCfg.NextProgramName");
	cfg->StringVar[i].Len = 20;

	i = varSTRING_curProgramName;
	strcpy(cfg->StringVar[i].enumTXT , "varSTRING_curProgramName");
		strcpy(cfg->StringVar[i].name, "Current Program Name");
	cfg->StringVar[i].pStr   = curCfg->CurProgramName;
	strcpy(cfg->StringVar[i].VarName , "CurCfg.CurProgramName");
	cfg->StringVar[i].Len = 20;

	/*
	i = varSTRING_WelProgramName;
	strcpy(cfg->StringVar[i].enumTXT , "varSTRING_WelProgramName");
	strcpy(cfg->StringVar[i].name, "Weld Program Name");
	cfg->StringVar[i].pStr = cfg->TXT_Resources[resWeldProgramName];
	strcpy(cfg->StringVar[i].VarName , "Cfg.TXT_Resources[7]");
	cfg->StringVar[i].Len = 15;
	strcpy(cfg->TXT_Resources[resWeldProgramName], "myFile000"); // temporary string for new save name

	i = varSTRING_Password;
	strcpy(cfg->StringVar[i].enumTXT , "varSTRING_Password");
	strcpy(cfg->StringVar[i].name, "Password ");
	cfg->StringVar[i].pStr	= m->Password;
	strcpy(cfg->StringVar[i].VarName , "Master[0].Password");
	cfg->StringVar[i].Len = 3;
	strcpy(m->Password , "000");
	*/

	for(i = varSTRING_HMI_0 ; i <= varSTRING_HMI_19 ; i++){
		xsprintf(cfg->StringVar[i].enumTXT , "varSTRING_HMI_%d" ,i - varSTRING_HMI_0 );
		xsprintf(cfg->StringVar[i].name, "HMI String Line_%d" ,i - varSTRING_HMI_0 );
		cfg->StringVar[i].pStr	= HMI_lines[ i - varSTRING_HMI_0];
		cfg->StringVar[i].Len   = 20;
		xsprintf(cfg->StringVar[i].VarName , "HMI_lines[%d]" , i - varSTRING_HMI_0);
	}

	i = varSTRING_UserName;
	strcpy(cfg->StringVar[i].enumTXT , "varSTRING_UserName");
	strcpy(cfg->StringVar[i].name , "User Name");
	cfg->StringVar[i].pStr	= UserName;
	strcpy(cfg->StringVar[i].VarName , "UserName");
	cfg->StringVar[i].Len = 20;

	i = varSTRING_PlcVersion;
	strcpy(cfg->StringVar[i].enumTXT , "varSTRING_PlcVersion");
	strcpy(cfg->StringVar[i].enumTXT , "PLC Program Version");
	cfg->StringVar[i].pStr = PLC_Version_TXT;
	strcpy(cfg->StringVar[i].VarName , "PLC_Version_TXT");
	cfg->StringVar[i].Len = 20;

	i = varSTRING_FileName;
	strcpy(cfg->StringVar[i].enumTXT , "varSTRING_FileName");
	strcpy(cfg->StringVar[i].name , "File Name");
	cfg->StringVar[i].pStr = File_RW.FileInfo[0].Filename;
	strcpy(cfg->StringVar[i].VarName , "File_RW.FileInfo[0].Filename");
	cfg->StringVar[i].Len = 20;

	i = varSTRING_MasteStepTXT;
	strcpy(cfg->StringVar[i].enumTXT , "varSTRING_MasteStepTXT");
	strcpy(cfg->StringVar[i].name , "Master State Machine Step");
	cfg->StringVar[i].pStr = m->sm.Text;
	strcpy(cfg->StringVar[i].VarName , "Master[0].sm.Text");
	cfg->StringVar[i].Len = 20;

	/////////////  Auto Indexing //////////////

	for(i = 0 ; i < m->paramIntgLastNum; i++)
		cfg->IntVar[i].Indx = i;

	for(i = 0 ; i < m->paramEnumLastNum; i++)
		cfg->EnumVar[i].Indx = i;

	for(i = 0 ; i < m->varLastNum; i++)
		var[i].Indx = i;

	for(i = 0 ; i < m->paramStrLastNum; i++)
		cfg->StringVar[i].Indx = i;

	// Text resources
	memcpy(cfg->TXT_Resources[resTXT_OSC_CAM] , CAM_TYPE_TXT , sizeof(CAM_TYPE_TXT));
	memcpy(cfg->TXT_Resources[resTXT_ON_OFF] , ON_OFF_TXT, sizeof(ON_OFF_TXT));
	memcpy(cfg->TXT_Resources[resWelProgramLinkMode] , JOBLINK_MODE_TXT, sizeof(JOBLINK_MODE_TXT));
	memcpy(cfg->TXT_Resources[resPathMode] , PATH_MODE_TXT, sizeof(PATH_MODE_TXT));
	memcpy(cfg->TXT_Resources[resWeldProgramCase] , JOB_CASE_TXT, sizeof(JOB_CASE_TXT));
	memcpy(cfg->TXT_Resources[resAVCMode] , AVC_MODE_TXT, sizeof(AVC_MODE_TXT));
	memcpy(cfg->TXT_Resources[resTIGMode] , TIG_MODE_TXT, sizeof(TIG_MODE_TXT));
	memcpy(cfg->TXT_Resources[resTVLMode] , TVL_MODE_TXT, sizeof(TVL_MODE_TXT));
	memcpy(cfg->TXT_Resources[resSYNCOption] , SYNCH_OPTION_TXT, sizeof(SYNCH_OPTION_TXT));
	memcpy(cfg->TXT_Resources[resTigCalMode] , TIG_CAL_MODE_TXT, sizeof(TIG_CAL_MODE_TXT));
	memcpy(cfg->TXT_Resources[resTXT_OSC_Mode] , OSC_MODE_TXT, sizeof(OSC_MODE_TXT));
	memcpy(cfg->TXT_Resources[resTXT_OSC_Synch] , OSC_SYNCH_TXT, sizeof(OSC_SYNCH_TXT));
	memcpy(cfg->TXT_Resources[resTXT_WF_AUX] , WF_AUX_TXT, sizeof(WF_AUX_TXT));

	/****************************/
	/*****  ERROR text ***********/

	strcpy(ErrorMgr.logs[ERROR_NONE].txt , " No Erros - Ready");

	/*
	strcpy(ErrorMgr.logs[ERROR_TML_1].txt , "TML1 :");
	strcpy(ErrorMgr.logs[ERROR_TML_2].txt , "TML2 :");
	strcpy(ErrorMgr.logs[ERROR_TML_3].txt , "TML3 :");
	strcpy(ErrorMgr.logs[ERROR_TML_4].txt , "TML4 :");
	strcpy(ErrorMgr.logs[ERROR_TML_5].txt , "TML5 :");
	strcpy(ErrorMgr.logs[ERROR_TML_6].txt , "TML6 :");
	strcpy(ErrorMgr.logs[ERROR_TML_7].txt , "TML7 :");
	strcpy(ErrorMgr.logs[ERROR_TML_8].txt , "TML8 :");
	strcpy(ErrorMgr.logs[ERROR_TML_9].txt , "TML9 :");
	strcpy(ErrorMgr.logs[ERROR_TML_10].txt , "TML10 :");

	strcpy(ErrorMgr.logs[ERROR_FATAL_TML_1].txt , "TML1 FATAL");
	strcpy(ErrorMgr.logs[ERROR_FATAL_TML_2].txt , "TML2 FATAL");
	strcpy(ErrorMgr.logs[ERROR_FATAL_TML_3].txt , "TML3 FATAL");
	strcpy(ErrorMgr.logs[ERROR_FATAL_TML_4].txt , "TML4 FATAL");
	strcpy(ErrorMgr.logs[ERROR_FATAL_TML_5].txt , "TML5 FATAL");
	strcpy(ErrorMgr.logs[ERROR_FATAL_TML_6].txt , "TML6 FATAL");
	strcpy(ErrorMgr.logs[ERROR_FATAL_TML_7].txt , "TML7 FATAL");
	strcpy(ErrorMgr.logs[ERROR_FATAL_TML_8].txt , "TML8 FATAL");
	strcpy(ErrorMgr.logs[ERROR_FATAL_TML_9].txt , "TML9 FATAL");
	strcpy(ErrorMgr.logs[ERROR_FATAL_TML_10].txt , "TML10 FATAL");

	strcpy(ErrorMgr.logs[ERROR_ACP_1].txt , "BR Axis #1");
	strcpy(ErrorMgr.logs[ERROR_ACP_2].txt , "BR Axis #2");
	strcpy(ErrorMgr.logs[ERROR_ACP_3].txt , "BR Axis #3");
	strcpy(ErrorMgr.logs[ERROR_ACP_4].txt , "BR Axis #4");
	strcpy(ErrorMgr.logs[ERROR_ACP_5].txt , "BR Axis #5");
	strcpy(ErrorMgr.logs[ERROR_ACP_6].txt , "BR Axis #6");
	strcpy(ErrorMgr.logs[ERROR_ACP_7].txt , "BR Axis #7");
	strcpy(ErrorMgr.logs[ERROR_ACP_8].txt , "BR Axis #8");

	strcpy(ErrorMgr.logs[ERROR_FATAL_ACP_1].txt , "Axis #1 ERR FATAL");
	strcpy(ErrorMgr.logs[ERROR_FATAL_ACP_2].txt , "Axis #2 ERR FATAL");
	strcpy(ErrorMgr.logs[ERROR_FATAL_ACP_3].txt , "Axis #3 ERR FATAL");
	strcpy(ErrorMgr.logs[ERROR_FATAL_ACP_4].txt , "Axis #4 ERR FATAL");
	strcpy(ErrorMgr.logs[ERROR_FATAL_ACP_5].txt , "Axis #5 ERR FATAL");
	strcpy(ErrorMgr.logs[ERROR_FATAL_ACP_6].txt , "ACP6 ERR FATAL");
	strcpy(ErrorMgr.logs[ERROR_FATAL_ACP_7].txt , "ACP7 ERR FATAL");
	strcpy(ErrorMgr.logs[ERROR_FATAL_ACP_8].txt , "ACP8 ERR FATAL");
	*/

	//strcpy(ErrorMgr.logs[ERROR_MOTOR_INIT].txt , "MTRS INIT TMO");

	//strcpy(ErrorMgr.logs[ERROR_ANGLE_NOT_EQ].txt , "ANGLE NOT SYNCHRO");

	strcpy(ErrorMgr.logs[ERROR_TIG_TOUCH_TMO].txt , "AVC TOUCH TMO");
	strcpy(ErrorMgr.logs[ERROR_TIG_SP_TMO].txt , 	"AVC VOLT TMO");
	strcpy(ErrorMgr.logs[ERROR_TIG_VOLT_ERR].txt , 	"AVC VOLT ERR");
	strcpy(ErrorMgr.logs[ERROR_TIG_AVC_LIMIT_ERR].txt , "AVC LIMITS ERR");

	strcpy(ErrorMgr.logs[ERROR_FILE_RW].txt , 	"File RW Err");

	strcpy(ErrorMgr.logs[ERROR_BR_HOME].txt , 	"BR Srv Home Err");

	strcpy(ErrorMgr.logs[ERROR_GAS_TMO].txt , 	"ARGON Tmo Err");

	strcpy(ErrorMgr.logs[ERROR_COOL_TMO].txt , 	"COOL Tmo Err");

	strcpy(ErrorMgr.logs[ERROR_TVL_STALL].txt ,  "TVL Stall Err");

	strcpy(ErrorMgr.logs[ERROR_TVL_STALL].txt ,  "TVL Stall Err");

	strcpy(ErrorMgr.logs[ERROR_ADROID_COM_LOST].txt ,  "Pendant Err");

	strcpy(ErrorMgr.logs[ERROR_ARCLINK_COM_LOST].txt ,  "ArcLink Com Lost");

	strcpy(ErrorMgr.logs[ERROR_ARCLINK_PS_ERR].txt ,  "ArcLink PS Err");

	strcpy(ErrorMgr.logs[ERROR_PROJECT_HRDW_ERR].txt ,  "WRONG CONTROLLER");

	strcpy(ErrorMgr.logs[ERROR_ESTOP_ERR].txt ,  "ESTOP !!!");

	strcpy(ErrorMgr.logs[ERROR_MODULE_ERR].txt ,  "MODULE MISSING");

	strcpy(ErrorMgr.logs[ERROR_TIG_MIG_SW_ERR].txt ,  "TIG/MIG Sw Err");

	//  Load Default Min Max for ENUM data

	for (i = 0 ; i < parENUM_LAST_PARAM; i++){

		curCfg->Param_ENUM[i].segmYes = 0;

		curCfg->Param_ENUM[i].incr = 1;
		curCfg->Param_ENUM[i].min = cfg->Param_ENUM[i].min;
		curCfg->Param_ENUM[i].max = cfg->Param_ENUM[i].max;

	}

	for (i = 0 ; i < parINT_LAST_PARAM; i++){

		if(curCfg->Param_INT[i].incr == 0)
			curCfg->Param_INT[i].incr = 1.0;

	}

	// Offset for File Manager

	File_RW._int.OffsetToWeldProgramRepeat = (UDINT)&File_RW.curCfgTemp.Param[parGEN_WeldProgramRepeat].val[0] - (UDINT)&File_RW.curCfgTemp;
	File_RW._int.OffsetToWeldProgramLinkMode = (UDINT)&File_RW.curCfgTemp.Param_ENUM[parENUM_WeldProgramLinkMode].val[0] - (UDINT)&File_RW.curCfgTemp;

	return;
}

void SetPageDict(PAGE_DICT_typ* dict , UINT indx , char* pTxt){

	if(dict){

		dict->indx = indx;
		strcpy(dict->enumTXT , pTxt);

	}

	return;

}

#endif
```

### Program Logical/FourAxisTigCtrl/Main2 (ANSIC) - Master program
